(* IEC 61131-3 sources: robocpp/validation/corpus/rejected, 7 files *)

(* ---- bad_access_path.st ---- *)
(* validation: feature=diagnostics.access-paths clause=2.4 *)
PROGRAM BadAccess
VAR_ACCESS
    PublicValue AT Missing : INT;
END_VAR
END_PROGRAM

(* ---- bad_assignment.st ---- *)
(* validation: feature=diagnostics.semantic clause=3.3 *)
PROGRAM BadAssignment
VAR
    Count : INT := 0;
END_VAR

Count := TRUE;
END_PROGRAM

(* ---- bad_call.st ---- *)
(* validation: feature=diagnostics.calls clause=2.5 *)
PROGRAM BadCall
VAR
    Out : INT := 0;
END_VAR

Out := ADD(IN1 := 1, Missing := 2);
END_PROGRAM

(* ---- bad_config.st ---- *)
(* validation: feature=diagnostics.configuration clause=2.7 *)
PROGRAM Worker
END_PROGRAM

CONFIGURATION BadPlant
RESOURCE Cpu ON PLC
    PROGRAM Main WITH MissingTask : Worker;
END_RESOURCE
END_CONFIGURATION

(* ---- bad_il_label.il ---- *)
(* validation: feature=diagnostics.il clause=3.2 *)
PROGRAM BadIlLabel
VAR
    Out : INT := 0;
END_VAR

JMP Missing
END_PROGRAM

(* ---- missing_end_program.st ---- *)
(* validation: feature=diagnostics.syntax clause=3.3 *)
PROGRAM MissingEnd
VAR
    Count : INT := 0;
END_VAR

Count := Count + 1;

(* ---- source_size_limit.st ---- *)
(* validation: feature=diagnostics.limits clause=limits *)
PROGRAM SourceSizeLimit
VAR
    ThisIdentifierIsIntentionallyTooLongForTheSmallValidationProfileAndKeepsGoingPastTheDefaultOneHundredTwentyEightCharacterLimitForTheCompilerReadinessCorpus : INT := 0;
END_VAR
END_PROGRAM
